TYPE ST_IOInput :
STRUCT
	IxAruIO AT%I*  :BOOL;
	xStartIO AT%I* :BOOL;
	xStopIO AT%I*  :BOOL;
	xResetIO AT%I* :BOOL;
	xAuto AT%I* : BOOL;
	xManual AT%I* : BOOL;
	
	
	
	iSetSpeedMotor : INT := 10;
	
	xAirPressureOk AT%I* : BOOL;
	
	//Btn in manual mode
	xHomingPosReached AT%I* : BOOL;
	xManualAct1GoIn AT%I* : BOOL;
	xManualAct1GoOut AT%I* : BOOL;
	
	//Btn in init mode
	xSetHomePos   AT%I*: BOOL;
	xJogXForward  AT%I*: BOOL;
	xJogYForward  AT%I*: BOOL;
	xJogXBackward AT%I*: BOOL;
	xJogYBackward AT%I*: BOOL;
	
	//Auto mode
	xAllowedGetPiece AT%I* : BOOL;
	xPiecePresent AT%I* : BOOL;
	xEmulateZDone AT%I* :Bool;
	
END_STRUCT
END_TYPE

(* stored: Version 1.1.0.1, ProductVersion 3.1.4020.12
   DUT ST_IOInput: Id {9cd39bb8-075d-45c1-8479-47b6e0b379ec} *)
